// TIA Portal V20 export
DATA_BLOCK "Hmi"   // DB199
// stored: MemoryReserve 100
   VAR
      mainHeader : Array[0.."NO_OF_PANELS"] of "LAF_typeHeader";   // Input from the status bar of the HMI
      operationInterlock : "LAF_typeOperationInterlockInterface";
   END_VAR
BEGIN
   mainHeader[0].plcToHmi.modeRequestsButtons.operatorControlAllowed := 16#003F;
   mainHeader[1].plcToHmi.stateCommandsButtons.visibility := 16#F;
   mainHeader[1].plcToHmi.stateCommandsButtons.operatorControlAllowed := 16#F;
   mainHeader[0].plcToHmi.specialFunctionButtons.visibility := 16#00330F7307337077;
   mainHeader[0].plcToHmi.specialFunctionButtons.operatorControlAllowed := 16#00330F7307337077;
END_DATA_BLOCK
